FUNCTION_BLOCK FB_AxisParameterSetExposed_Test EXTENDS FB_MotorTestSuite
(*
    Quick Check to verify exposed NC parameters are copied properly.
*)
VAR
    stMotionStage: ST_MotionStage;
    fbMotionStage: FB_MotionStage;
    nTestCounter: UINT;
    bOneTestDone: BOOL;
    tonTimer: TON;
END_VAR

IF nTestCounter = 0 THEN
    nTestCounter := 1;
END_IF

// Test that parameters are copied to the exposed parameters properly.
TestParameterCopy(1);

IF bOneTestDone THEN
    bOneTestDone := FALSE;
    nTestCounter := nTestCounter + 1;
    tonTimer(IN:=FALSE);
END_IF;

// Use this timer to time out any tests that stall
tonTimer(
    IN:=nTestCounter >= 1,
    PT:=T#2s,
);

METHOD TestParameterCopy
VAR_INPUT
    nTestIndex: UINT;
END_VAR
VAR_INST
    bLocalInit: BOOL := TRUE;
    bAllModified: BOOL;
    bReady: BOOL;
    bDone: BOOL;
END_VAR
TEST(CONCAT('TestParameterCopy', UINT_TO_STRING(nTestIndex)));
IF nTestCounter <> nTestIndex OR bOneTestDone THEN
    RETURN;
END_IF

fbMotionStage(stMotionStage:=stMotionStage);

IF bLocalInit THEN
    stMotionStage.stAxisParametersExposed.bCtrlEnablePosDiffControl     := 100;
    stMotionStage.stAxisParametersExposed.bEncEnableSoftEndMaxControl   := 101;
    stMotionStage.stAxisParametersExposed.bEncEnableSoftEndMinControl   := 102;
    stMotionStage.stAxisParametersExposed.fAccelerationMax              := 103;
    stMotionStage.stAxisParametersExposed.fCtrlPosDiffMax               := 104;
    stMotionStage.stAxisParametersExposed.fCtrlPosDiffMaxTime           := 105;
    stMotionStage.stAxisParametersExposed.fDecelerationMax              := 106;
    stMotionStage.stAxisParametersExposed.fEncSoftEndMax                := 107;
    stMotionStage.stAxisParametersExposed.fEncSoftEndMin                := 108;
    stMotionStage.stAxisParametersExposed.fVeloMaximum                  := 109;

    bLocalInit := FALSE;

    bAllModified :=
        stMotionStage.stAxisParametersExposed.bCtrlEnablePosDiffControl     <> stMotionStage.stAxisParameters.bCtrlEnablePosDiffControl AND
        stMotionStage.stAxisParametersExposed.bEncEnableSoftEndMaxControl   <> stMotionStage.stAxisParameters.bEncEnableSoftEndMaxControl AND
        stMotionStage.stAxisParametersExposed.bEncEnableSoftEndMinControl   <> stMotionStage.stAxisParameters.bEncEnableSoftEndMinControl AND
        stMotionStage.stAxisParametersExposed.fAccelerationMax              <> stMotionStage.stAxisParameters.fAccelerationMax AND
        stMotionStage.stAxisParametersExposed.fCtrlPosDiffMax               <> stMotionStage.stAxisParameters.fCtrlPosDiffMax AND
        stMotionStage.stAxisParametersExposed.fCtrlPosDiffMaxTime           <> stMotionStage.stAxisParameters.fCtrlPosDiffMaxTime AND
        stMotionStage.stAxisParametersExposed.fDecelerationMax              <> stMotionStage.stAxisParameters.fDecelerationMax AND
        stMotionStage.stAxisParametersExposed.fEncSoftEndMax                <> stMotionStage.stAxisParameters.fEncSoftEndMax AND
        stMotionStage.stAxisParametersExposed.fEncSoftEndMin                <> stMotionStage.stAxisParameters.fEncSoftEndMin AND
        stMotionStage.stAxisParametersExposed.fVeloMaximum                  <> stMotionStage.stAxisParameters.fVeloMaximum;

    AssertTrue(
        Condition:=bAllModified,
        Message:='One or more parameters was not modified initially so the check is invalid.',
    );
END_IF

bReady :=
        stMotionStage.stAxisParameters.bCtrlEnablePosDiffControl     <> 0 AND
        stMotionStage.stAxisParameters.bEncEnableSoftEndMaxControl   <> 0 AND
        stMotionStage.stAxisParameters.bEncEnableSoftEndMinControl   <> 0 AND
        stMotionStage.stAxisParameters.fAccelerationMax              <> 0 AND
        stMotionStage.stAxisParameters.fCtrlPosDiffMax               <> 0 AND
        stMotionStage.stAxisParameters.fCtrlPosDiffMaxTime           <> 0 AND
        stMotionStage.stAxisParameters.fDecelerationMax              <> 0 AND
        stMotionStage.stAxisParameters.fEncSoftEndMax                <> 0 AND
        stMotionStage.stAxisParameters.fEncSoftEndMin                <> 0 AND
        stMotionStage.stAxisParameters.fVeloMaximum                  <> 0;

IF bReady THEN
    bDone :=
        stMotionStage.stAxisParametersExposed.bCtrlEnablePosDiffControl     = stMotionStage.stAxisParameters.bCtrlEnablePosDiffControl AND
        stMotionStage.stAxisParametersExposed.bEncEnableSoftEndMaxControl   = stMotionStage.stAxisParameters.bEncEnableSoftEndMaxControl AND
        stMotionStage.stAxisParametersExposed.bEncEnableSoftEndMinControl   = stMotionStage.stAxisParameters.bEncEnableSoftEndMinControl AND
        stMotionStage.stAxisParametersExposed.fAccelerationMax              = stMotionStage.stAxisParameters.fAccelerationMax AND
        stMotionStage.stAxisParametersExposed.fCtrlPosDiffMax               = stMotionStage.stAxisParameters.fCtrlPosDiffMax AND
        stMotionStage.stAxisParametersExposed.fCtrlPosDiffMaxTime           = stMotionStage.stAxisParameters.fCtrlPosDiffMaxTime AND
        stMotionStage.stAxisParametersExposed.fDecelerationMax              = stMotionStage.stAxisParameters.fDecelerationMax AND
        stMotionStage.stAxisParametersExposed.fEncSoftEndMax                = stMotionStage.stAxisParameters.fEncSoftEndMax AND
        stMotionStage.stAxisParametersExposed.fEncSoftEndMin                = stMotionStage.stAxisParameters.fEncSoftEndMin AND
        stMotionStage.stAxisParametersExposed.fVeloMaximum                  = stMotionStage.stAxisParameters.fVeloMaximum;
END_IF

IF bDone OR tonTimer.Q THEN
    AssertFalse(
        Condition:=tonTimer.Q,
        Message:=CONCAT(CONCAT('Failed to update the parameters within ', TIME_TO_STRING(tonTimer.PT)),' seconds.'),
    );
    AssertTrue(
        Condition:=bDone,
        Message:='One or more parameters was not copied properly.',
    );

    bOneTestDone := TRUE;
    TEST_FINISHED();
END_IF
END_METHOD

END_FUNCTION_BLOCK

(* stored: Version 1.1.0.1
   POU FB_AxisParameterSetExposed_Test: Id {862cf200-7f25-43c6-8605-e66b08e38db7}, SpecialFunc None
   Method TestParameterCopy: Id {7caa7a7e-60eb-46a7-b83a-472b67bef094} *)
